TYPE ST_Values_Checked_Iosys :
STRUCT
	sTimestamp			: STRING(255);						//Timestamp
	sId					: STRING(255);						//Id from the Datapoint
	lrValue				: LREAL;							//Value from Datapoint
END_STRUCT
END_TYPE

(* stored: Version 1.1.0.1, ProductVersion 3.1.4024.9
   DUT ST_Values_Checked_Iosys: Id {159de91d-1fb4-478a-a625-e6b71add1200} *)
